FUNCTION_BLOCK Producer
  (* Standard: 61499-2 *)
  (* Version 0.1, 2017-00-09, hpea485, UOA *)
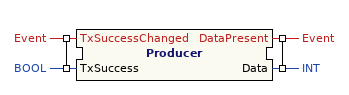
  EVENT_INPUT
    TxSuccessChanged WITH TxSuccess;
  END_EVENT
  EVENT_OUTPUT
    DataPresent WITH Data;
  END_EVENT
  VAR_INPUT
    TxSuccess : BOOL;
  END_VAR
  VAR_OUTPUT
    Data : INT;
  END_VAR
  VAR
    Count : INT := 0;
  END_VAR
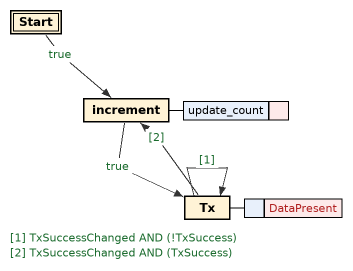
  EC_STATES
    Start;
    increment : update_count;
    Tx : -> DataPresent;
  END_STATES
  EC_TRANSITIONS
    Start TO increment := true;
    increment TO Tx := true;
    Tx TO increment := TxSuccessChanged AND (TxSuccess);
    Tx TO Tx := TxSuccessChanged AND (!TxSuccess);
  END_TRANSITIONS
  ALGORITHM update_count IN C:
me->Count++;
me->Data = me->Count;
  END_ALGORITHM
END_FUNCTION_BLOCK
